VAR_GLOBAL
	Digital_Input AT %I* : ARRAY [1..10] OF BOOL;
END_VAR

(* stored: Version 1.1.0.1, ProductVersion 3.1.0.36
   GVL IO_DigiIn_GVL: Id {f05251e0-ccf8-4838-98d9-dc6f2fa872b8} *)
